// TIA Portal V20 export
FUNCTION_BLOCK "FB_Alarms"   // FB300, SCL
{ S7_Optimized_Access := 'FALSE' }
// stored: AutoNumber false, SetENOAutomatically false
   VAR
      sAlarmsLevel0 : Bool;
      sAlarmsLevel1 : Bool;
      sAlarmsLevel2 : Bool;
      sAlarmsLevel3 : Bool;
      sAlarmsLevel4 : Bool;
      sAlarmsLevel5 : Bool;
      sAlarmsLevel6 : Bool;
      sRTBuzzer { S7_SetPoint := 'True'} : R_TRIG;
      sActiveBuzzer : Bool;
      sTableInParkPosition : Bool;
   END_VAR
   VAR_TEMP
      tIndexRID : Int;
   END_VAR
BEGIN
   REGION Description header 
       //==================================================================================
       // POSALUX Swiss SA / (C) Copyright 2024
       //----------------------------------------------------------------------------------
       // Title: Alarmes_Machine
       // Comment/Function: Alarm management block for the machine, organized by severity
       //                   levels (0 to 6).
       //                   Each level triggers specific actions. Alarms are grouped by
       //                   their levels.
       // Author: Gowsigan SRITHARAN
       // Engineering: TIA Portal v17
       //----------------------------------------------------------------------------------
       // Change log table:
       // Version  | Date     | Expert in charge | Changes applied
       // ---------|----------|------------------|------------------------------------
       // 00.00.01 | 20241206 | GSR              | First released version
       // ---------|----------|------------------|------------------------------------
       // ==================================================================================
   END_REGION
   REGION "Alarm" level 0
       // Messages
       #sAlarmsLevel0 :=
       "LBP_AlarmMsgs".UserA[00].A70UUxx[35]

       OR "LBP_AlarmMsgs".UserA[02].A70UUxx[36]

       OR "LBP_AlarmMsgs".UserA[05].A70UUxx[32]
       OR "LBP_AlarmMsgs".UserA[05].A70UUxx[33]
       OR "LBP_AlarmMsgs".UserA[05].A70UUxx[34]
       OR "LBP_AlarmMsgs".UserA[05].A70UUxx[35]
       OR "LBP_AlarmMsgs".UserA[05].A70UUxx[36]
       OR "LBP_AlarmMsgs".UserA[05].A70UUxx[37]
       OR "LBP_AlarmMsgs".UserA[05].A70UUxx[38]
       OR "LBP_AlarmMsgs".UserA[05].A70UUxx[39]
       OR "LBP_AlarmMsgs".UserA[05].A70UUxx[42]
       OR "LBP_AlarmMsgs".UserA[05].A70UUxx[48]
       OR "LBP_AlarmMsgs".UserA[05].A70UUxx[50]
       OR "LBP_AlarmMsgs".UserA[05].A70UUxx[51]

       OR "LBP_AlarmMsgs".UserA[08].A70UUxx[00]
       OR "LBP_AlarmMsgs".UserA[08].A70UUxx[41]

       OR "LBP_AlarmMsgs".ChanA[1].RID_5C02xx[00]
       OR "LBP_AlarmMsgs".ChanA[1].RID_5C02xx[01]
       OR "LBP_AlarmMsgs".ChanA[1].RID_5C02xx[02]
       OR "LBP_AlarmMsgs".ChanA[1].RID_5C02xx[03]
       OR "LBP_AlarmMsgs".ChanA[1].RID_5C02xx[04]
       OR "LBP_AlarmMsgs".ChanA[1].RID_5C02xx[05]
       OR "LBP_AlarmMsgs".ChanA[1].RID_5C02xx[06]
       OR "LBP_AlarmMsgs".ChanA[1].RID_5C02xx[07]
       OR "LBP_AlarmMsgs".ChanA[1].RID_5C02xx[08]
       OR "LBP_AlarmMsgs".ChanA[1].RID_5C02xx[09]
       OR "LBP_AlarmMsgs".ChanA[1].RID_5C02xx[10]
       OR "LBP_AlarmMsgs".ChanA[1].RID_5C02xx[11]
       OR "LBP_AlarmMsgs".ChanA[1].RID_5C02xx[12]
       OR "LBP_AlarmMsgs".ChanA[1].RID_5C02xx[13]
       OR "LBP_AlarmMsgs".ChanA[1].RID_5C02xx[14]
       OR "LBP_AlarmMsgs".ChanA[1].RID_5C02xx[15];
   END_REGION

   REGION "Alarm" level 1
       // Blinking blue light + user acknowledge
       #sAlarmsLevel1 :=
          "LBP_AlarmMsgs".UserA[00].A70UUxx[59]
       OR "LBP_AlarmMsgs".UserA[00].A70UUxx[60]
       OR "LBP_AlarmMsgs".UserA[00].A70UUxx[61]
       OR "LBP_AlarmMsgs".UserA[00].A70UUxx[62]

       OR "LBP_AlarmMsgs".UserA[03].A70UUxx[48]

       OR "LBP_AlarmMsgs".UserA[04].A70UUxx[41]
       OR "LBP_AlarmMsgs".UserA[04].A70UUxx[42]

       OR "LBP_AlarmMsgs".UserA[05].A70UUxx[43]

       OR "LBP_AlarmMsgs".UserA[06].A70UUxx[62]
       OR "LBP_AlarmMsgs".UserA[06].A70UUxx[63]

       OR "LBP_AlarmMsgs".UserA[30].A70UUxx[32]
       OR "LBP_AlarmMsgs".UserA[30].A70UUxx[33]
       OR "LBP_AlarmMsgs".UserA[30].A70UUxx[34]
       OR "LBP_AlarmMsgs".UserA[30].A70UUxx[35]
       OR "LBP_AlarmMsgs".UserA[30].A70UUxx[36]
       OR "LBP_AlarmMsgs".UserA[30].A70UUxx[37]
       OR "LBP_AlarmMsgs".UserA[30].A70UUxx[38]
       OR "LBP_AlarmMsgs".UserA[30].A70UUxx[39]
       OR "LBP_AlarmMsgs".UserA[30].A70UUxx[10]
       OR "LBP_AlarmMsgs".UserA[30].A70UUxx[41]
       OR "LBP_AlarmMsgs".UserA[30].A70UUxx[42]
       OR "LBP_AlarmMsgs".UserA[30].A70UUxx[43]
       OR "LBP_AlarmMsgs".UserA[30].A70UUxx[44]
       OR "LBP_AlarmMsgs".UserA[30].A70UUxx[45]
       OR "LBP_AlarmMsgs".UserA[30].A70UUxx[46]
       OR "LBP_AlarmMsgs".UserA[30].A70UUxx[47];
   END_REGION

   REGION "Alarm" level 2
       // blinking blue light and red beacon + user acknowledge
       #sAlarmsLevel2 :=
       "LBP_AlarmMsgs".UserA[00].A70UUxx[55]
       OR "LBP_AlarmMsgs".UserA[00].A70UUxx[63]

       OR "LBP_AlarmMsgs".UserA[04].A70UUxx[03]
       OR "LBP_AlarmMsgs".UserA[04].A70UUxx[04]
       OR "LBP_AlarmMsgs".UserA[04].A70UUxx[05]
       OR "LBP_AlarmMsgs".UserA[04].A70UUxx[06]
       OR "LBP_AlarmMsgs".UserA[04].A70UUxx[20]
       OR "LBP_AlarmMsgs".UserA[04].A70UUxx[21]
       OR "LBP_AlarmMsgs".UserA[04].A70UUxx[22]
       OR "LBP_AlarmMsgs".UserA[04].A70UUxx[23]

       OR "LBP_AlarmMsgs".UserA[05].A70UUxx[08]
       OR "LBP_AlarmMsgs".UserA[05].A70UUxx[09]
       OR "LBP_AlarmMsgs".UserA[05].A70UUxx[10]
       OR "LBP_AlarmMsgs".UserA[05].A70UUxx[11]
       OR "LBP_AlarmMsgs".UserA[05].A70UUxx[12]

       OR "LBP_AlarmMsgs".UserA[06].A70UUxx[52]
       OR "LBP_AlarmMsgs".UserA[06].A70UUxx[53]

       OR "LBP_AlarmMsgs".UserA[07].A70UUxx[00]
       OR "LBP_AlarmMsgs".UserA[07].A70UUxx[01]
       OR "LBP_AlarmMsgs".UserA[07].A70UUxx[02]
       OR "LBP_AlarmMsgs".UserA[07].A70UUxx[03]
       OR "LBP_AlarmMsgs".UserA[07].A70UUxx[04]
       OR "LBP_AlarmMsgs".UserA[07].A70UUxx[05]
       OR "LBP_AlarmMsgs".UserA[07].A70UUxx[06]
       OR "LBP_AlarmMsgs".UserA[07].A70UUxx[07]
       OR "LBP_AlarmMsgs".UserA[07].A70UUxx[08]
       OR "LBP_AlarmMsgs".UserA[07].A70UUxx[09]
       OR "LBP_AlarmMsgs".UserA[07].A70UUxx[10]
       OR "LBP_AlarmMsgs".UserA[07].A70UUxx[11]
       OR "LBP_AlarmMsgs".UserA[07].A70UUxx[40]
       OR "LBP_AlarmMsgs".UserA[07].A70UUxx[41]
       OR "LBP_AlarmMsgs".UserA[07].A70UUxx[42]
       OR "LBP_AlarmMsgs".UserA[07].A70UUxx[43]
       OR "LBP_AlarmMsgs".UserA[07].A70UUxx[44]
       OR "LBP_AlarmMsgs".UserA[07].A70UUxx[45]
       OR "LBP_AlarmMsgs".UserA[07].A70UUxx[46]
       OR "LBP_AlarmMsgs".UserA[07].A70UUxx[47]
       OR "LBP_AlarmMsgs".UserA[07].A70UUxx[48]
       OR "LBP_AlarmMsgs".UserA[07].A70UUxx[49]
       OR "LBP_AlarmMsgs".UserA[07].A70UUxx[50]
       OR "LBP_AlarmMsgs".UserA[07].A70UUxx[51]
       OR "LBP_AlarmMsgs".UserA[07].A70UUxx[52]
       OR "LBP_AlarmMsgs".UserA[07].A70UUxx[53]
       OR "LBP_AlarmMsgs".UserA[07].A70UUxx[54]
       OR "LBP_AlarmMsgs".UserA[07].A70UUxx[55]
       OR "LBP_AlarmMsgs".UserA[07].A70UUxx[56]
       OR "LBP_AlarmMsgs".UserA[07].A70UUxx[57]
       OR "LBP_AlarmMsgs".UserA[07].A70UUxx[58]
       OR "LBP_AlarmMsgs".UserA[07].A70UUxx[59]
       OR "LBP_AlarmMsgs".UserA[07].A70UUxx[60]
       OR "LBP_AlarmMsgs".UserA[07].A70UUxx[61]

       OR "LBP_AlarmMsgs".UserA[30].A70UUxx[00]
       OR "LBP_AlarmMsgs".UserA[30].A70UUxx[01]
       OR "LBP_AlarmMsgs".UserA[30].A70UUxx[02]
       OR "LBP_AlarmMsgs".UserA[30].A70UUxx[03]
       OR "LBP_AlarmMsgs".UserA[30].A70UUxx[04]
       OR "LBP_AlarmMsgs".UserA[30].A70UUxx[05]
       OR "LBP_AlarmMsgs".UserA[30].A70UUxx[06]
       OR "LBP_AlarmMsgs".UserA[30].A70UUxx[07]
       OR "LBP_AlarmMsgs".UserA[30].A70UUxx[08]
       OR "LBP_AlarmMsgs".UserA[30].A70UUxx[09]
       OR "LBP_AlarmMsgs".UserA[30].A70UUxx[10]
       OR "LBP_AlarmMsgs".UserA[30].A70UUxx[11]
       OR "LBP_AlarmMsgs".UserA[30].A70UUxx[12]
       OR "LBP_AlarmMsgs".UserA[30].A70UUxx[13]
       OR "LBP_AlarmMsgs".UserA[30].A70UUxx[14]
       OR "LBP_AlarmMsgs".UserA[30].A70UUxx[15];
   END_REGION

   REGION "Alarm" level 3
       // blinking blue light and red beacon + stop program at next step + user acknowledge
       #sAlarmsLevel3 :=
       "LBP_AlarmMsgs".UserA[00].A70UUxx[06]
       OR "LBP_AlarmMsgs".UserA[00].A70UUxx[07]
       OR "LBP_AlarmMsgs".UserA[00].A70UUxx[08]
       OR "LBP_AlarmMsgs".UserA[00].A70UUxx[14]
       OR "LBP_AlarmMsgs".UserA[00].A70UUxx[15]

       OR "LBP_AlarmMsgs".UserA[01].A70UUxx[03]
       OR "LBP_AlarmMsgs".UserA[01].A70UUxx[04]
       OR "LBP_AlarmMsgs".UserA[01].A70UUxx[05]
       OR "LBP_AlarmMsgs".UserA[01].A70UUxx[06]
       OR "LBP_AlarmMsgs".UserA[01].A70UUxx[07]
       OR "LBP_AlarmMsgs".UserA[01].A70UUxx[08]
       OR "LBP_AlarmMsgs".UserA[01].A70UUxx[09]
       OR "LBP_AlarmMsgs".UserA[01].A70UUxx[10]
       OR "LBP_AlarmMsgs".UserA[01].A70UUxx[11]
       OR "LBP_AlarmMsgs".UserA[01].A70UUxx[12]
       OR "LBP_AlarmMsgs".UserA[01].A70UUxx[13]
       OR "LBP_AlarmMsgs".UserA[01].A70UUxx[14]
       OR "LBP_AlarmMsgs".UserA[01].A70UUxx[15]
       OR "LBP_AlarmMsgs".UserA[01].A70UUxx[20]

       OR "LBP_AlarmMsgs".UserA[02].A70UUxx[00]
       OR "LBP_AlarmMsgs".UserA[02].A70UUxx[01]
       OR "LBP_AlarmMsgs".UserA[02].A70UUxx[02]
       OR "LBP_AlarmMsgs".UserA[02].A70UUxx[04]
       OR "LBP_AlarmMsgs".UserA[02].A70UUxx[05]
       OR "LBP_AlarmMsgs".UserA[02].A70UUxx[06]
       //   OR "LBP_AlarmMsgs".UserA[02].A70UUxx[07]
       //   OR "LBP_AlarmMsgs".UserA[02].A70UUxx[08]
       //   OR "LBP_AlarmMsgs".UserA[02].A70UUxx[09]
       //   OR "LBP_AlarmMsgs".UserA[02].A70UUxx[10]
       //   OR "LBP_AlarmMsgs".UserA[02].A70UUxx[11]
       //   OR "LBP_AlarmMsgs".UserA[02].A70UUxx[12]
       // OR "LBP_AlarmMsgs".UserA[02].A70UUxx[18]
       OR "LBP_AlarmMsgs".UserA[02].A70UUxx[19]
       OR "LBP_AlarmMsgs".UserA[02].A70UUxx[20]
       OR "LBP_AlarmMsgs".UserA[02].A70UUxx[21]
       OR "LBP_AlarmMsgs".UserA[02].A70UUxx[22]

       OR "LBP_AlarmMsgs".UserA[03].A70UUxx[15]
       OR "LBP_AlarmMsgs".UserA[03].A70UUxx[16]
       OR "LBP_AlarmMsgs".UserA[03].A70UUxx[17]
       OR "LBP_AlarmMsgs".UserA[03].A70UUxx[18]
       OR "LBP_AlarmMsgs".UserA[03].A70UUxx[19]
       OR "LBP_AlarmMsgs".UserA[03].A70UUxx[20]
       OR "LBP_AlarmMsgs".UserA[03].A70UUxx[21]
       OR "LBP_AlarmMsgs".UserA[03].A70UUxx[22]
       OR "LBP_AlarmMsgs".UserA[03].A70UUxx[23]
       OR "LBP_AlarmMsgs".UserA[03].A70UUxx[24]
       OR "LBP_AlarmMsgs".UserA[03].A70UUxx[25]
       OR "LBP_AlarmMsgs".UserA[03].A70UUxx[26]
       OR "LBP_AlarmMsgs".UserA[03].A70UUxx[27]
       OR "LBP_AlarmMsgs".UserA[03].A70UUxx[28]
     //  OR "LBP_AlarmMsgs".UserA[03].A70UUxx[29] WFA Msg défaut BW Loader, pas d'acquit nécéssaire

       OR "LBP_AlarmMsgs".UserA[04].A70UUxx[09]
       OR "LBP_AlarmMsgs".UserA[04].A70UUxx[10]
       OR "LBP_AlarmMsgs".UserA[04].A70UUxx[24]
       OR "LBP_AlarmMsgs".UserA[04].A70UUxx[25]
       OR "LBP_AlarmMsgs".UserA[04].A70UUxx[26]
       OR "LBP_AlarmMsgs".UserA[04].A70UUxx[27]
       OR "LBP_AlarmMsgs".UserA[04].A70UUxx[28]
       OR "LBP_AlarmMsgs".UserA[04].A70UUxx[29]

       OR "LBP_AlarmMsgs".UserA[06].A70UUxx[04]
       OR "LBP_AlarmMsgs".UserA[06].A70UUxx[05]
       OR "LBP_AlarmMsgs".UserA[06].A70UUxx[06]
       OR "LBP_AlarmMsgs".UserA[06].A70UUxx[07]
       OR "LBP_AlarmMsgs".UserA[06].A70UUxx[08]
    //   OR "LBP_AlarmMsgs".UserA[06].A70UUxx[09]
       OR "LBP_AlarmMsgs".UserA[06].A70UUxx[10]
     //  OR "LBP_AlarmMsgs".UserA[06].A70UUxx[11]
       OR "LBP_AlarmMsgs".UserA[06].A70UUxx[40]
       OR "LBP_AlarmMsgs".UserA[06].A70UUxx[41]
       OR "LBP_AlarmMsgs".UserA[06].A70UUxx[50]
     //  OR "LBP_AlarmMsgs".UserA[06].A70UUxx[51]
       OR "LBP_AlarmMsgs".UserA[06].A70UUxx[54]
       OR "LBP_AlarmMsgs".UserA[06].A70UUxx[55]
       // OR "LBP_AlarmMsgs".UserA[06].A70UUxx[56]
       OR "LBP_AlarmMsgs".UserA[06].A70UUxx[57]
       //  OR "LBP_AlarmMsgs".UserA[06].A70UUxx[58]
       OR "LBP_AlarmMsgs".UserA[06].A70UUxx[59]
       OR "LBP_AlarmMsgs".UserA[06].A70UUxx[60]
      // OR "LBP_AlarmMsgs".UserA[06].A70UUxx[61]

       // OR "LBP_AlarmMsgs".UserA[08].A70UUxx[08]
       OR "LBP_AlarmMsgs".UserA[08].A70UUxx[09]
       OR "LBP_AlarmMsgs".UserA[08].A70UUxx[10]
       OR "LBP_AlarmMsgs".UserA[08].A70UUxx[11]
       //  OR "LBP_AlarmMsgs".UserA[08].A70UUxx[12]
       OR "LBP_AlarmMsgs".UserA[08].A70UUxx[13]
       OR "LBP_AlarmMsgs".UserA[08].A70UUxx[14]
       OR "LBP_AlarmMsgs".UserA[08].A70UUxx[15]
       OR "LBP_AlarmMsgs".UserA[08].A70UUxx[16]
       OR "LBP_AlarmMsgs".UserA[08].A70UUxx[17]
       // OR "LBP_AlarmMsgs".UserA[08].A70UUxx[20]
       // OR "LBP_AlarmMsgs".UserA[08].A70UUxx[21]
       OR "LBP_AlarmMsgs".UserA[08].A70UUxx[22]
       // OR "LBP_AlarmMsgs".UserA[08].A70UUxx[23]
       OR "LBP_AlarmMsgs".UserA[08].A70UUxx[24];

   END_REGION

   REGION "Alarm" level 4
       // blinking blue light and red beacon + stop program at next step + acknowledge by reset button
       #sAlarmsLevel4 :=
          "LBP_AlarmMsgs".UserA[00].A70UUxx[02]
       OR "LBP_AlarmMsgs".UserA[00].A70UUxx[05]

       OR "LBP_AlarmMsgs".UserA[05].A70UUxx[01]
       OR "LBP_AlarmMsgs".UserA[05].A70UUxx[02]

    //   OR "LBP_AlarmMsgs".UserA[06].A70UUxx[42]
       OR "LBP_AlarmMsgs".UserA[06].A70UUxx[43]
    //   OR "LBP_AlarmMsgs".UserA[06].A70UUxx[44]
       OR "LBP_AlarmMsgs".UserA[06].A70UUxx[45]
       OR "LBP_AlarmMsgs".UserA[06].A70UUxx[46]
       OR "LBP_AlarmMsgs".UserA[06].A70UUxx[47]
     //  OR "LBP_AlarmMsgs".UserA[06].A70UUxx[48]
       OR "LBP_AlarmMsgs".UserA[06].A70UUxx[49];
   END_REGION

   REGION "Alarm" level 5
       // blinking blue light and red beacon + acknowledge by reset button + power off
       #sAlarmsLevel5 :=
          "LBP_AlarmMsgs".UserA[00].A70UUxx[03]
      // OR "LBP_AlarmMsgs".UserA[00].A70UUxx[04] WFA 20251205 

       // OR "LBP_AlarmMsgs".UserA[03].A70UUxx[30]
       // OR "LBP_AlarmMsgs".UserA[03].A70UUxx[31]

       OR "LBP_AlarmMsgs".UserA[05].A70UUxx[00]

       OR "LBP_AlarmMsgs".UserA[06].A70UUxx[00]
       OR "LBP_AlarmMsgs".UserA[06].A70UUxx[01]
     // OR "LBP_AlarmMsgs".UserA[06].A70UUxx[02] WFA 20251118 - A revoir temp min axe
       OR "LBP_AlarmMsgs".UserA[06].A70UUxx[03]
       OR "LBP_AlarmMsgs".UserA[06].A70UUxx[23]
       OR "LBP_AlarmMsgs".UserA[06].A70UUxx[25];
   END_REGION

   REGION "Alarm" level 6
       // Power off and shut down
       #sAlarmsLevel6 :=
          "LBP_AlarmMsgs".UserA[04].A70UUxx[02];
   END_REGION

   REGION Buzzer management
       IF #sRTBuzzer.Q THEN
           #sActiveBuzzer := TRUE;
       ELSIF "DB_McpKeyboardSignals".sAlarmReset.sKeySWStatus OR "MCP1_In".reset THEN
           #sActiveBuzzer := FALSE;
       END_IF;

       "DB_DigitalOutputs".sBuzzerActivation.sSWStatus :=
       #sActiveBuzzer
       OR "DB_McpKeyboardSignals".sLightTest.sKeySWStatus; //Test Lampes-LED
   END_REGION

   REGION Ack alarm level 0
       IF "DB_McpKeyboardSignals".sAlarmReset.sKeySWStatus OR "MCP1_In".reset THEN
           "LBP_AlarmMsgs".UserA[00].A70UUxx[35] := FALSE;

           "LBP_AlarmMsgs".UserA[02].A70UUxx[36] := FALSE;

           "LBP_AlarmMsgs".UserA[05].A70UUxx[32] := FALSE;
           "LBP_AlarmMsgs".UserA[05].A70UUxx[33] := FALSE;
           "LBP_AlarmMsgs".UserA[05].A70UUxx[34] := FALSE;
           "LBP_AlarmMsgs".UserA[05].A70UUxx[35] := FALSE;
           "LBP_AlarmMsgs".UserA[05].A70UUxx[36] := FALSE;
           "LBP_AlarmMsgs".UserA[05].A70UUxx[37] := FALSE;
           "LBP_AlarmMsgs".UserA[05].A70UUxx[38] := FALSE;
           "LBP_AlarmMsgs".UserA[05].A70UUxx[39] := FALSE;
           "LBP_AlarmMsgs".UserA[05].A70UUxx[42] := FALSE;
           "LBP_AlarmMsgs".UserA[05].A70UUxx[48] := FALSE;
           "LBP_AlarmMsgs".UserA[05].A70UUxx[50] := FALSE;
           "LBP_AlarmMsgs".UserA[05].A70UUxx[51] := FALSE;

           "LBP_AlarmMsgs".UserA[08].A70UUxx[00] := FALSE;
           "LBP_AlarmMsgs".UserA[08].A70UUxx[41] := FALSE;
       END_IF;
   END_REGION

   REGION Ack alarm level 1
       IF "DB_McpKeyboardSignals".sAlarmReset.sKeySWStatus OR "MCP1_In".reset THEN
           "LBP_AlarmMsgs".UserA[00].A70UUxx[59] := FALSE;
           "LBP_AlarmMsgs".UserA[00].A70UUxx[61] := FALSE;
           "LBP_AlarmMsgs".UserA[00].A70UUxx[62] := FALSE;

           "LBP_AlarmMsgs".UserA[04].A70UUxx[41] := FALSE;
           "LBP_AlarmMsgs".UserA[04].A70UUxx[42] := FALSE;

           "LBP_AlarmMsgs".UserA[05].A70UUxx[43] := FALSE;

           "LBP_AlarmMsgs".UserA[06].A70UUxx[62] := FALSE;
           "LBP_AlarmMsgs".UserA[06].A70UUxx[63] := FALSE;

           "LBP_AlarmMsgs".UserA[30].A70UUxx[32] := FALSE;
           "LBP_AlarmMsgs".UserA[30].A70UUxx[33] := FALSE;
           "LBP_AlarmMsgs".UserA[30].A70UUxx[34] := FALSE;
           "LBP_AlarmMsgs".UserA[30].A70UUxx[35] := FALSE;
           "LBP_AlarmMsgs".UserA[30].A70UUxx[36] := FALSE;
           "LBP_AlarmMsgs".UserA[30].A70UUxx[37] := FALSE;
           "LBP_AlarmMsgs".UserA[30].A70UUxx[38] := FALSE;
           "LBP_AlarmMsgs".UserA[30].A70UUxx[39] := FALSE;
           "LBP_AlarmMsgs".UserA[30].A70UUxx[10] := FALSE;
           "LBP_AlarmMsgs".UserA[30].A70UUxx[41] := FALSE;
           "LBP_AlarmMsgs".UserA[30].A70UUxx[42] := FALSE;
           "LBP_AlarmMsgs".UserA[30].A70UUxx[43] := FALSE;
           "LBP_AlarmMsgs".UserA[30].A70UUxx[44] := FALSE;
           "LBP_AlarmMsgs".UserA[30].A70UUxx[45] := FALSE;
           "LBP_AlarmMsgs".UserA[30].A70UUxx[46] := FALSE;
           "LBP_AlarmMsgs".UserA[30].A70UUxx[47] := FALSE;
       END_IF;
   END_REGION

   REGION Ack alarm level 2
       IF "DB_McpKeyboardSignals".sAlarmReset.sKeySWStatus OR "MCP1_In".reset THEN
           "LBP_AlarmMsgs".UserA[00].A70UUxx[63] := FALSE;

           "LBP_AlarmMsgs".UserA[04].A70UUxx[03] := FALSE;
           "LBP_AlarmMsgs".UserA[04].A70UUxx[04] := FALSE;
           "LBP_AlarmMsgs".UserA[04].A70UUxx[05] := FALSE;
           "LBP_AlarmMsgs".UserA[04].A70UUxx[06] := FALSE;
           "LBP_AlarmMsgs".UserA[04].A70UUxx[20] := FALSE;
           "LBP_AlarmMsgs".UserA[04].A70UUxx[21] := FALSE;
           "LBP_AlarmMsgs".UserA[04].A70UUxx[22] := FALSE;
           "LBP_AlarmMsgs".UserA[04].A70UUxx[23] := FALSE;

           "LBP_AlarmMsgs".UserA[05].A70UUxx[08] := FALSE;
           "LBP_AlarmMsgs".UserA[05].A70UUxx[09] := FALSE;
           "LBP_AlarmMsgs".UserA[05].A70UUxx[10] := FALSE;
           "LBP_AlarmMsgs".UserA[05].A70UUxx[11] := FALSE;
           "LBP_AlarmMsgs".UserA[05].A70UUxx[12] := FALSE;

           "LBP_AlarmMsgs".UserA[06].A70UUxx[52] := FALSE;
           "LBP_AlarmMsgs".UserA[06].A70UUxx[53] := FALSE;

           "LBP_AlarmMsgs".UserA[07].A70UUxx[00] := FALSE;
           "LBP_AlarmMsgs".UserA[07].A70UUxx[01] := FALSE;
           "LBP_AlarmMsgs".UserA[07].A70UUxx[02] := FALSE;
           "LBP_AlarmMsgs".UserA[07].A70UUxx[03] := FALSE;
           "LBP_AlarmMsgs".UserA[07].A70UUxx[04] := FALSE;
           "LBP_AlarmMsgs".UserA[07].A70UUxx[05] := FALSE;
           "LBP_AlarmMsgs".UserA[07].A70UUxx[06] := FALSE;
           "LBP_AlarmMsgs".UserA[07].A70UUxx[07] := FALSE;
           "LBP_AlarmMsgs".UserA[07].A70UUxx[08] := FALSE;
           "LBP_AlarmMsgs".UserA[07].A70UUxx[09] := FALSE;
           "LBP_AlarmMsgs".UserA[07].A70UUxx[10] := FALSE;
           "LBP_AlarmMsgs".UserA[07].A70UUxx[11] := FALSE;
           "LBP_AlarmMsgs".UserA[07].A70UUxx[40] := FALSE;
           "LBP_AlarmMsgs".UserA[07].A70UUxx[41] := FALSE;
           "LBP_AlarmMsgs".UserA[07].A70UUxx[42] := FALSE;
           "LBP_AlarmMsgs".UserA[07].A70UUxx[43] := FALSE;
           "LBP_AlarmMsgs".UserA[07].A70UUxx[44] := FALSE;
           "LBP_AlarmMsgs".UserA[07].A70UUxx[45] := FALSE;
           "LBP_AlarmMsgs".UserA[07].A70UUxx[46] := FALSE;
           "LBP_AlarmMsgs".UserA[07].A70UUxx[47] := FALSE;
           "LBP_AlarmMsgs".UserA[07].A70UUxx[48] := FALSE;
           "LBP_AlarmMsgs".UserA[07].A70UUxx[49] := FALSE;
           "LBP_AlarmMsgs".UserA[07].A70UUxx[50] := FALSE;
           "LBP_AlarmMsgs".UserA[07].A70UUxx[51] := FALSE;
           "LBP_AlarmMsgs".UserA[07].A70UUxx[52] := FALSE;
           "LBP_AlarmMsgs".UserA[07].A70UUxx[53] := FALSE;
           "LBP_AlarmMsgs".UserA[07].A70UUxx[54] := FALSE;
           "LBP_AlarmMsgs".UserA[07].A70UUxx[55] := FALSE;
           "LBP_AlarmMsgs".UserA[07].A70UUxx[56] := FALSE;
           "LBP_AlarmMsgs".UserA[07].A70UUxx[57] := FALSE;
           "LBP_AlarmMsgs".UserA[07].A70UUxx[58] := FALSE;
           "LBP_AlarmMsgs".UserA[07].A70UUxx[59] := FALSE;
           "LBP_AlarmMsgs".UserA[07].A70UUxx[60] := FALSE;
           "LBP_AlarmMsgs".UserA[07].A70UUxx[61] := FALSE;

           "LBP_AlarmMsgs".UserA[30].A70UUxx[00] := FALSE;
           "LBP_AlarmMsgs".UserA[30].A70UUxx[01] := FALSE;
           "LBP_AlarmMsgs".UserA[30].A70UUxx[02] := FALSE;
           "LBP_AlarmMsgs".UserA[30].A70UUxx[03] := FALSE;
           "LBP_AlarmMsgs".UserA[30].A70UUxx[04] := FALSE;
           "LBP_AlarmMsgs".UserA[30].A70UUxx[05] := FALSE;
           "LBP_AlarmMsgs".UserA[30].A70UUxx[06] := FALSE;
           "LBP_AlarmMsgs".UserA[30].A70UUxx[07] := FALSE;
           "LBP_AlarmMsgs".UserA[30].A70UUxx[08] := FALSE;
           "LBP_AlarmMsgs".UserA[30].A70UUxx[09] := FALSE;
           "LBP_AlarmMsgs".UserA[30].A70UUxx[10] := FALSE;
           "LBP_AlarmMsgs".UserA[30].A70UUxx[11] := FALSE;
           "LBP_AlarmMsgs".UserA[30].A70UUxx[12] := FALSE;
           "LBP_AlarmMsgs".UserA[30].A70UUxx[13] := FALSE;
           "LBP_AlarmMsgs".UserA[30].A70UUxx[14] := FALSE;
           "LBP_AlarmMsgs".UserA[30].A70UUxx[15] := FALSE;
       END_IF;
   END_REGION

   REGION Ack alarm level 3
       IF "DB_McpKeyboardSignals".sAlarmReset.sKeySWStatus OR "MCP1_In".reset THEN
           "LBP_AlarmMsgs".UserA[00].A70UUxx[06] := FALSE;
           "LBP_AlarmMsgs".UserA[00].A70UUxx[07] := FALSE;
           "LBP_AlarmMsgs".UserA[00].A70UUxx[08] := FALSE;
           "LBP_AlarmMsgs".UserA[00].A70UUxx[14] := FALSE;
           "LBP_AlarmMsgs".UserA[00].A70UUxx[15] := FALSE;

           "LBP_AlarmMsgs".UserA[01].A70UUxx[03] := FALSE;
           "LBP_AlarmMsgs".UserA[01].A70UUxx[04] := FALSE;
           "LBP_AlarmMsgs".UserA[01].A70UUxx[05] := FALSE;
           "LBP_AlarmMsgs".UserA[01].A70UUxx[06] := FALSE;
           "LBP_AlarmMsgs".UserA[01].A70UUxx[07] := FALSE;
           "LBP_AlarmMsgs".UserA[01].A70UUxx[08] := FALSE;
           "LBP_AlarmMsgs".UserA[01].A70UUxx[09] := FALSE;
           "LBP_AlarmMsgs".UserA[01].A70UUxx[10] := FALSE;
           "LBP_AlarmMsgs".UserA[01].A70UUxx[11] := FALSE;
           "LBP_AlarmMsgs".UserA[01].A70UUxx[12] := FALSE;
           "LBP_AlarmMsgs".UserA[01].A70UUxx[13] := FALSE;
           "LBP_AlarmMsgs".UserA[01].A70UUxx[14] := FALSE;
           "LBP_AlarmMsgs".UserA[01].A70UUxx[15] := FALSE;
           "LBP_AlarmMsgs".UserA[01].A70UUxx[20] := FALSE;

           "LBP_AlarmMsgs".UserA[02].A70UUxx[00] := FALSE;
           "LBP_AlarmMsgs".UserA[02].A70UUxx[01] := FALSE;
           "LBP_AlarmMsgs".UserA[02].A70UUxx[02] := FALSE;
           "LBP_AlarmMsgs".UserA[02].A70UUxx[04] := FALSE;
           "LBP_AlarmMsgs".UserA[02].A70UUxx[05] := FALSE;
           "LBP_AlarmMsgs".UserA[02].A70UUxx[06] := FALSE;
           "LBP_AlarmMsgs".UserA[02].A70UUxx[07] := FALSE;
           "LBP_AlarmMsgs".UserA[02].A70UUxx[08] := FALSE;
           "LBP_AlarmMsgs".UserA[02].A70UUxx[09] := FALSE;
           "LBP_AlarmMsgs".UserA[02].A70UUxx[10] := FALSE;
           "LBP_AlarmMsgs".UserA[02].A70UUxx[11] := FALSE;
           "LBP_AlarmMsgs".UserA[02].A70UUxx[12] := FALSE;
           "LBP_AlarmMsgs".UserA[02].A70UUxx[18] := FALSE;
           "LBP_AlarmMsgs".UserA[02].A70UUxx[19] := FALSE;
           "LBP_AlarmMsgs".UserA[02].A70UUxx[20] := FALSE;
           "LBP_AlarmMsgs".UserA[02].A70UUxx[21] := FALSE;
           "LBP_AlarmMsgs".UserA[02].A70UUxx[22] := FALSE;

           "LBP_AlarmMsgs".UserA[03].A70UUxx[15] := FALSE;
           "LBP_AlarmMsgs".UserA[03].A70UUxx[16] := FALSE;
           "LBP_AlarmMsgs".UserA[03].A70UUxx[17] := FALSE;
           "LBP_AlarmMsgs".UserA[03].A70UUxx[18] := FALSE;
           "LBP_AlarmMsgs".UserA[03].A70UUxx[19] := FALSE;
           "LBP_AlarmMsgs".UserA[03].A70UUxx[20] := FALSE;
           "LBP_AlarmMsgs".UserA[03].A70UUxx[21] := FALSE;
           "LBP_AlarmMsgs".UserA[03].A70UUxx[22] := FALSE;
           "LBP_AlarmMsgs".UserA[03].A70UUxx[23] := FALSE;
           "LBP_AlarmMsgs".UserA[03].A70UUxx[24] := FALSE;
           "LBP_AlarmMsgs".UserA[03].A70UUxx[25] := FALSE;
           "LBP_AlarmMsgs".UserA[03].A70UUxx[26] := FALSE;
           "LBP_AlarmMsgs".UserA[03].A70UUxx[27] := FALSE;
           "LBP_AlarmMsgs".UserA[03].A70UUxx[28] := FALSE;
           "LBP_AlarmMsgs".UserA[03].A70UUxx[29] := FALSE;

           "LBP_AlarmMsgs".UserA[04].A70UUxx[09] := FALSE;
           "LBP_AlarmMsgs".UserA[04].A70UUxx[10] := FALSE;
           "LBP_AlarmMsgs".UserA[04].A70UUxx[24] := FALSE;
           "LBP_AlarmMsgs".UserA[04].A70UUxx[25] := FALSE;
           "LBP_AlarmMsgs".UserA[04].A70UUxx[26] := FALSE;
           "LBP_AlarmMsgs".UserA[04].A70UUxx[27] := FALSE;
           "LBP_AlarmMsgs".UserA[04].A70UUxx[28] := FALSE;
           "LBP_AlarmMsgs".UserA[04].A70UUxx[29] := FALSE;

           "LBP_AlarmMsgs".UserA[06].A70UUxx[04] := FALSE;
           "LBP_AlarmMsgs".UserA[06].A70UUxx[05] := FALSE;
           "LBP_AlarmMsgs".UserA[06].A70UUxx[06] := FALSE;
           "LBP_AlarmMsgs".UserA[06].A70UUxx[07] := FALSE;
           "LBP_AlarmMsgs".UserA[06].A70UUxx[08] := FALSE;
           "LBP_AlarmMsgs".UserA[06].A70UUxx[09] := FALSE;
           "LBP_AlarmMsgs".UserA[06].A70UUxx[10] := FALSE;
           "LBP_AlarmMsgs".UserA[06].A70UUxx[11] := FALSE;
           "LBP_AlarmMsgs".UserA[06].A70UUxx[40] := FALSE;
           "LBP_AlarmMsgs".UserA[06].A70UUxx[41] := FALSE;
           "LBP_AlarmMsgs".UserA[06].A70UUxx[50] := FALSE;
           "LBP_AlarmMsgs".UserA[06].A70UUxx[51] := FALSE;
           "LBP_AlarmMsgs".UserA[06].A70UUxx[54] := FALSE;
           "LBP_AlarmMsgs".UserA[06].A70UUxx[55] := FALSE;
           "LBP_AlarmMsgs".UserA[06].A70UUxx[56] := FALSE;
           "LBP_AlarmMsgs".UserA[06].A70UUxx[57] := FALSE;
           "LBP_AlarmMsgs".UserA[06].A70UUxx[58] := FALSE;
           "LBP_AlarmMsgs".UserA[06].A70UUxx[59] := FALSE;
           "LBP_AlarmMsgs".UserA[06].A70UUxx[60] := FALSE;
           "LBP_AlarmMsgs".UserA[06].A70UUxx[61] := FALSE;

           "LBP_AlarmMsgs".UserA[08].A70UUxx[08] := FALSE;
           "LBP_AlarmMsgs".UserA[08].A70UUxx[09] := FALSE;
           "LBP_AlarmMsgs".UserA[08].A70UUxx[10] := FALSE;
           "LBP_AlarmMsgs".UserA[08].A70UUxx[11] := FALSE;
           "LBP_AlarmMsgs".UserA[08].A70UUxx[12] := FALSE;
           "LBP_AlarmMsgs".UserA[08].A70UUxx[13] := FALSE;
           "LBP_AlarmMsgs".UserA[08].A70UUxx[14] := FALSE;
           "LBP_AlarmMsgs".UserA[08].A70UUxx[15] := FALSE;
           "LBP_AlarmMsgs".UserA[08].A70UUxx[16] := FALSE;
           "LBP_AlarmMsgs".UserA[08].A70UUxx[17] := FALSE;

           "LBP_AlarmMsgs".UserA[08].A70UUxx[20] := FALSE;
           "LBP_AlarmMsgs".UserA[08].A70UUxx[21] := FALSE;
           "LBP_AlarmMsgs".UserA[08].A70UUxx[22] := FALSE;
           "LBP_AlarmMsgs".UserA[08].A70UUxx[23] := FALSE;
           "LBP_AlarmMsgs".UserA[08].A70UUxx[24] := FALSE;
       END_IF;
   END_REGION

   REGION Ack alarm level 4
       IF "MCP1_In".reset THEN
           "LBP_AlarmMsgs".UserA[00].A70UUxx[02] := FALSE;
           "LBP_AlarmMsgs".UserA[00].A70UUxx[05] := FALSE;

           "LBP_AlarmMsgs".UserA[05].A70UUxx[01] := FALSE;
           "LBP_AlarmMsgs".UserA[05].A70UUxx[02] := FALSE;

           "LBP_AlarmMsgs".UserA[06].A70UUxx[42] := FALSE;
           "LBP_AlarmMsgs".UserA[06].A70UUxx[43] := FALSE;
           "LBP_AlarmMsgs".UserA[06].A70UUxx[44] := FALSE;
           "LBP_AlarmMsgs".UserA[06].A70UUxx[45] := FALSE;
           "LBP_AlarmMsgs".UserA[06].A70UUxx[46] := FALSE;
           "LBP_AlarmMsgs".UserA[06].A70UUxx[47] := FALSE;
           "LBP_AlarmMsgs".UserA[06].A70UUxx[48] := FALSE;
           "LBP_AlarmMsgs".UserA[06].A70UUxx[49] := FALSE;
       END_IF;
   END_REGION

   REGION Ack alarm level 5
       IF "MCP1_In".reset THEN
           "LBP_AlarmMsgs".UserA[00].A70UUxx[03] := FALSE;
           "LBP_AlarmMsgs".UserA[00].A70UUxx[04] := FALSE;

           "LBP_AlarmMsgs".UserA[03].A70UUxx[30] := FALSE;
           "LBP_AlarmMsgs".UserA[03].A70UUxx[31] := FALSE;

           "LBP_AlarmMsgs".UserA[05].A70UUxx[00] := FALSE;

           "LBP_AlarmMsgs".UserA[06].A70UUxx[00] := FALSE;
           "LBP_AlarmMsgs".UserA[06].A70UUxx[01] := FALSE;
           "LBP_AlarmMsgs".UserA[06].A70UUxx[02] := FALSE;
           "LBP_AlarmMsgs".UserA[06].A70UUxx[03] := FALSE;
           "LBP_AlarmMsgs".UserA[06].A70UUxx[23] := FALSE;
           "LBP_AlarmMsgs".UserA[06].A70UUxx[25] := FALSE;
       END_IF;
   END_REGION

   REGION Ack alarm level 6
       IF "MCP1_In".reset THEN
           "LBP_AlarmMsgs".UserA[04].A70UUxx[02] := FALSE;
       END_IF;
   END_REGION

   REGION Ack alarm RID 5102xx
       IF "LBP_Chan1".E_ChanReset THEN
           "LBP_AlarmMsgs".ChanA[1].RID_5C02xx[00] := FALSE;
           "LBP_AlarmMsgs".ChanA[1].RID_5C02xx[01] := FALSE;
           "LBP_AlarmMsgs".ChanA[1].RID_5C02xx[02] := FALSE;
           "LBP_AlarmMsgs".ChanA[1].RID_5C02xx[03] := FALSE;
           "LBP_AlarmMsgs".ChanA[1].RID_5C02xx[04] := FALSE;
           "LBP_AlarmMsgs".ChanA[1].RID_5C02xx[05] := FALSE;
           "LBP_AlarmMsgs".ChanA[1].RID_5C02xx[06] := FALSE;
           "LBP_AlarmMsgs".ChanA[1].RID_5C02xx[07] := FALSE;
           "LBP_AlarmMsgs".ChanA[1].RID_5C02xx[08] := FALSE;
           "LBP_AlarmMsgs".ChanA[1].RID_5C02xx[09] := FALSE;
           "LBP_AlarmMsgs".ChanA[1].RID_5C02xx[10] := FALSE;
           "LBP_AlarmMsgs".ChanA[1].RID_5C02xx[11] := FALSE;
           "LBP_AlarmMsgs".ChanA[1].RID_5C02xx[12] := FALSE;
           "LBP_AlarmMsgs".ChanA[1].RID_5C02xx[13] := FALSE;
           "LBP_AlarmMsgs".ChanA[1].RID_5C02xx[14] := FALSE;
           "LBP_AlarmMsgs".ChanA[1].RID_5C02xx[15] := FALSE;
       END_IF;
   END_REGION
END_FUNCTION_BLOCK
